{attribute 'linkalways'} 
{attribute 'no_explicit_call' := 'This FB is a CLASS and must be accessed using methods or properties'}
{attribute 'enable_dynamic_creation'}
FUNCTION_BLOCK _TOD EXTENDS DatatypeBase
VAR
	localData : TOD;
	activeData : REFERENCE TO TOD REF= localData;
END_VAR

PROPERTY PUBLIC Address : PVOID
GET
Address := ADR(activeData);
END_GET
END_PROPERTY

METHOD PUBLIC ClearReference
VAR_INPUT
END_VAR
activeData REF= localData;
END_METHOD

METHOD PUBLIC Clone : I_Datatype
VAR
    pClone : POINTER TO _TOD;
END_VAR
pClone := __NEW(_TOD(InitialValue := Value));
Clone := pClone^;
END_METHOD

METHOD FB_init : BOOL
VAR_INPUT
	bInitRetains : BOOL; // if TRUE, the retain variables are initialized (warm start / cold start)
	bInCopyCode : BOOL;  // if TRUE, the instance afterwards gets moved WORDo the copy code (online change)
	InitialValue : TOD;
END_VAR
localData := InitialValue;
END_METHOD

PROPERTY PUBLIC IecType : T_MAXSTRING
GET
IecType := 'TOD';
END_GET
END_PROPERTY

METHOD PUBLIC MakeReferenceTo
VAR_INPUT
	ReferenceTarget : REFERENCE TO TOD;
END_VAR
activeData REF= ReferenceTarget;
END_METHOD

METHOD PUBLIC SerializeWith
VAR_INPUT
	Serializer : I_Serializer;
END_VAR
Serializer.AddTod(activeData);
END_METHOD

PROPERTY PUBLIC Size : UDINT
GET
Size := SIZEOF(activeData);
END_GET
END_PROPERTY

METHOD TryDeserializeFrom : BOOL
VAR_INPUT
	Deserializer : I_Deserializer;
	Feedback : I_DeserializerFeedback;
END_VAR
TryDeserializeFrom := Deserializer.TryGetTod(activeData, Feedback);
END_METHOD

METHOD TryMakeReferenceTo : BOOL
VAR_INPUT
	Target : I_Datatype;
END_VAR
VAR
	pTargetData : POINTER TO TOD;
END_VAR
IF NOT (Target.IecType = IecType) THEN
	RETURN;
END_IF

pTargetData := Target.Address;
activeData REF= pTargetData^;
TryMakeReferenceTo := TRUE;
END_METHOD

PROPERTY PUBLIC Value : TOD
GET
Value := activeData;
END_GET
SET
activeData := Value;
END_SET
END_PROPERTY

END_FUNCTION_BLOCK

(* stored: Version 1.1.0.1, ProductVersion 3.1.4024.12
   POU _TOD: Id {52bd5b26-6ad5-0a51-382c-4dbd3487f46c}, SpecialFunc None
   Folder Constructor: Id {710e214e-6868-0d3d-2168-fd2c43da2339}
   Property Address: Id {b678ada3-d73b-0df5-3247-414a4bfdd231}
   Get Get: Id {421a083f-7889-0416-1a8a-c32b15c46cf0}
   Method ClearReference: Id {f77e43b0-5319-0dc2-3f2d-b2a27762232f}
   Method Clone: Id {bcf68f09-1024-0f2d-2b1e-961720a8981a}
   Method FB_init: Id {3fab4cdc-0c76-03fb-203f-fd524cb45261}
   Property IecType: Id {465d04b7-af87-04b5-3c6a-0216f2c60e66}
   Get Get: Id {e657eff8-8375-0d47-2f89-b9bc1fce380e}
   Method MakeReferenceTo: Id {cb7a25f8-ec2e-08cd-3949-e1d2b92b448d}
   Method SerializeWith: Id {586b1cc7-a831-09db-2a94-1d85bbe43635}
   Property Size: Id {534d91c2-d2fc-0142-3869-37913b882b43}
   Get Get: Id {f97749d6-ec2b-0869-141f-9186685008a2}
   Method TryDeserializeFrom: Id {b2f1aebe-aab3-0d82-094b-2892b7c8975c}
   Method TryMakeReferenceTo: Id {6186bb35-9ca1-0204-1a78-652320292fef}
   Property Value: Id {3773c9c0-b562-0f63-16c9-3e235b3bb967}
   Get Get: Id {3dd8fd8b-4e10-0c0a-2169-210a172d2206}
   Set Set: Id {692b59d4-7ae7-021f-294d-c3003e1d7480} *)
